{attribute 'GeneratedUsingTerminal: EL6851-0010-0016'}
{attribute addProperty BoxType "EL6851-0010-0016"}
{attribute addProperty Id "DMX_StatusAT %I*DMX_Status_5ECDEABE8DMX_Channel_1_64AT %I*DMX_Channel_005FDEFD64WcStateAT %I*WcState_9091E0EB2InfoDataAT %I*InfoData_32EB74EA10"}
{attribute addProperty CRC "699107392"}
{attribute addProperty Size "84"}
TYPE EL6851_29AB8840 EXTENDS EtcSlaveTerminalBase_947E5A46 :
STRUCT
	{attribute addProperty Name "DMX_Status"}
	DMX_Status : DMX_Status_5ECDEABE;
	{attribute addProperty Name "DMX_Channel_1_64"}
	DMX_Channel_1_64 : DMX_Channel_005FDEFD;
	{attribute addProperty Name "WcState"}
	WcState : WcState_9091E0EB;
	{attribute addProperty Name "InfoData"}
	InfoData : InfoData_32EB74EA;
END_STRUCT
END_TYPE

(* stored: Version 1.2.0.0, ProductVersion 3.1.4024.9
   DUT EL6851_29AB8840: Id {710813ef-fe1d-4c60-8cd5-2ae8b22dab51} *)
